(* IEC 61131-3 sources: digital-academy-template-provatest/src, 2 files *)

(* ---- deviatore.st ---- *)
USING Tipi;

NAMESPACE Libreria

    CLASS deviatore

        VAR PUBLIC
            ID :INT;
            sensore : BOOL; // il sensore del deviatore del magazzino rosso si attiva se vede un pacco rosso
            cntrlApri : BOOL; // segnale per aprire il deviatore (se è aperto lascia passare i pacchi)
            cntrlChiudi : BOOL; // segnale per chiudere il deviatore (se è chiuso devia i pacchi)
            chiuso : BOOL;
        END_VAR

        METHOD PUBLIC Init // inizializzazione del deviatore
            VAR_INPUT
                IDinit : INT;
            END_VAR
            ID:=IDinit;
            sensore := FALSE; // all'inizio non vede il pacco
            chiuso := FALSE; // all'inizio il deviatore è aperto
            cntrlApri := FALSE;
            cntrlChiudi := FALSE; // all'inizio non ci sono comandi di apertura o chiusura
        END_METHOD

        METHOD PUBLIC ChiudiDeviatore // nel main se (sensore = TRUE) vogliamo chiudere il deviatore
            cntrlChiudi := TRUE;
            cntrlApri := FALSE;
        END_METHOD // NB ci pensa test.st a definire (chiuso := TRUE)

        METHOD PUBLIC ApriDeviatore // una volta deviato il pacco nel mai (sensore = FALSE) vogliamo aprire il deviatore
            cntrlApri := TRUE;
            cntrlChiudi := FALSE;
        END_METHOD // NB ci pensa test.st a definire (chiuso := FALSE)

    END_CLASS

END_NAMESPACE

(* ---- MainProgram.st ---- *)
USING tipi;
USING Libreria;

PROGRAM MainProgram

    VAR
        n_mag : INT:=3; // numero magazzini
        nastri : ARRAY[1..3] OF nastro;
        deviatori : ARRAY[1..3] OF deviatore;
        magazzini : ARRAY[1..3+1] OF magazzino;
        PLCinizializzato : BOOL := FALSE; // il PLC va inizializzato solo una volta altrimenti il test non funziona
    END_VAR

    VAR_TEMP
        i:INT;
    END_VAR

    IF NOT PLCinizializzato THEN // il PLC va inizializzato solo una volta altrimenti il test non funziona
        FOR i := 1 TO n_mag DO // inizializzare componenti
            nastri[i].Init(i);
            deviatori[i].Init(i);
            magazzini[i].Init(i);
        END_FOR;
        magazzini[n_mag+1].Init(n_mag+1); //inizializzazione magazzino scarti

        PLCinizializzato := TRUE; // il PLC è stato inizializzato
    END_IF;

    FOR i := 1 TO n_mag DO

        // controllo del deviatore
        IF deviatori[i].sensore = TRUE AND deviatori[i].chiuso = FALSE THEN
            deviatori[i].ChiudiDeviatore();
        ELSIF deviatori[i].sensore = FALSE AND deviatori[i].chiuso = TRUE THEN
            deviatori[i].ApriDeviatore();
        END_IF;

    END_FOR;

END_PROGRAM
